(*
SPDX-FileCopyrightText: © 2026 Oleksandr Tiutyk <trofimich@gmail.com>
SPDX-License-Identifier: MIT
License: https://opensource.org/license/mit
*)

(*!
<summary>Loads file contents through cyclic task execution.</summary>
<description>
The native FB_FileLoad opens the file in binary mode, reads the requested byte count and closes it. Its
documented path support is the addressed target's local filesystem, not a network-share path. Use one owner
task. Configure FilePath, AmsNetId, TargetBuffer, TargetBufferSize and Timeout before Start and keep them
unchanged until STOPPED. The caller supplies live writable memory of at least TargetBufferSize bytes and
retains it through stopping after failure or cancellation. Do not access that memory concurrently with the
operation. Missing path, null buffer and zero size are rejected during execution; capacity and pointer
lifetime cannot be verified by this wrapper. Native errors use Task failure handling. Continue Execute until
STOPPED. Cancellation drains pending work without restoring buffer contents. WORK_DONE means the native
request completed without an error; this wrapper does not compare the returned byte count with file size or
promise a complete snapshot of a concurrently modified file. LoadedBytesCount exposes the result only after
STOPPED and WORK_DONE. Reset preserves configuration.
</description>
*)

{attribute 'no_explicit_call' := 'do not call this function block directly'}
FUNCTION_BLOCK LoadFile EXTENDS TOF_Tasks.Task IMPLEMENTS IFileSystemTask
VAR_STAT
	//! <summary>Static type metadata available before the base task initializes its default name.</summary>
	{attribute 'hide'}
	_ClassName : STRING := __POUNAME();
END_VAR
VAR
    _LoadFile : Tc2_System.FB_FileLoad; 
END_VAR

(*!
<summary>Selects the ADS target for the native filesystem operation.</summary>
<description>
Configure before Start and keep unchanged until STOPPED; the setter stores configuration without submitting
I/O.
</description>
*)
{attribute 'monitoring' := 'call'}
PROPERTY AmsNetId : Tc2_System.T_AmsNetID
GET
AmsNetId := _LoadFile.sNetId;
END_GET
SET
_LoadFile.sNetId := AmsNetId;
END_SET
END_PROPERTY

(*!
<summary>Provides the concrete type name used in diagnostics.</summary>
<description>
Returns borrowed read-only metadata; keep the instance alive and do not modify the referenced string.
Initialized static storage is ready during base Task.FB_init; this getter has no side effects or exceptions.
</description>
*)
{attribute 'monitoring' := 'call'}
PROPERTY ClassName : REFERENCE TO STRING
GET
ClassName REF= _ClassName;
END_GET
END_PROPERTY

(*!
<summary>Provides the configured path for the file operation.</summary>
<description>
The setter copies text without performing I/O. Configure before Start and keep unchanged until STOPPED; Reset
preserves it. The native service determines whether the path is usable.
</description>
*)
{attribute 'monitoring' := 'call'}
PROPERTY FilePath : Tc2_System.T_MaxString
GET
FilePath := _LoadFile.sPathName;
END_GET
SET
_LoadFile.sPathName := FilePath;
END_SET
END_PROPERTY

(*!
<summary>Reports the byte count from a successfully completed load.</summary>
<description>
Returns the native result only while State.Stopped and FinalStopReason.WorkDone are both TRUE. In every other
state, including READY, RUNNING, failure and cancellation, returns the initial value of the property type.
This default is not a success indicator; inspect the task state and final reason. Zero outside successful
completion does not mean the target buffer was unchanged. The getter does not modify native outputs or
buffers. Copy a successful result before Reset or reuse.
</description>
*)
{attribute 'monitoring' := 'call'}
PROPERTY LoadedBytesCount : UDINT
GET
IF NOT State.Stopped OR_ELSE NOT FinalStopReason.WorkDone THEN
	RETURN;
END_IF

LoadedBytesCount := _LoadFile.cbRead;
END_GET
END_PROPERTY

(*!
<summary>Provides the library namespace used in diagnostics.</summary>
<description>Returns borrowed read-only namespace storage; do not modify the referenced string.</description>
*)
{attribute 'monitoring' := 'call'}
PROPERTY NamespaceName : REFERENCE TO STRING
GET
NamespaceName REF= CurrentNamespace.Name;
END_GET
END_PROPERTY

(*!
<summary>Resets the native request edge after the task has stopped.</summary>
<description>
Preserves configured inputs and does not undo completed filesystem effects. Pending I/O must finish during
stopping before this hook runs.
</description>
*)
METHOD PROTECTED OnReset
_LoadFile(bExecute := FALSE);
END_METHOD

(*!
<summary>Submits and advances a native file load into caller-owned memory.</summary>
<description>
Validates required configuration before submitting the request. Native errors raise an exception for the base
Task failure/stopping path without dynamic string-builder allocations. Normal completion reports DONE only
after the native block is no longer busy. No rollback is performed.
</description>
<param name="processingState">BUSY while pending; DONE after native completion without an error.</param>
<param name="stopReasonMessage">Not changed here; failures are passed through exceptions.</param>
*)
METHOD PROTECTED OnRunning
VAR_OUTPUT
	processingState : TOF_Tasks.TASK_PROCESSING_STATE;
END_VAR
VAR_IN_OUT
	stopReasonMessage : TOF_Core.ERROR_MESSAGE;
END_VAR
VAR
	formattedExceptionMessage : TOF_Core.ERROR_MESSAGE;
END_VAR
IF NOT _LoadFile.bExecute THEN 
	IF TOF_Core.Strings.IsNullOrWhiteSpace(stringToCheck := _LoadFile.sPathName) THEN
		TOF_Core.Exceptions.ThrowDataMemberNotSpecified(
			sourceNamespaceName := NamespaceName,
			sourceClassName := ClassName,
			sourcePOUName := __POUNAME(),
			sourcePosition := __POSITION(),
			dataMemberName := 'FilePath'
		);		
	END_IF

	IF _LoadFile.pReadBuff = 0 THEN
		TOF_Core.Exceptions.ThrowDataMemberNotSpecified(
			sourceNamespaceName := NamespaceName,
			sourceClassName := ClassName,
			sourcePOUName := __POUNAME(),
			sourcePosition := __POSITION(),
			dataMemberName := 'TargetBuffer'
		);		
	END_IF

	IF _LoadFile.cbReadLen = 0 THEN
		TOF_Core.Exceptions.ThrowDataMemberNotSpecified(
			sourceNamespaceName := NamespaceName,
			sourceClassName := ClassName,
			sourcePOUName := __POUNAME(),
			sourcePosition := __POSITION(),
			dataMemberName := 'TargetBufferSize'
		);		
	END_IF
END_IF

_LoadFile(bExecute := TRUE);

IF _LoadFile.bError THEN
	TOF_Core.WideStrings.Append255(
		formattedExceptionMessage,
		"An error occurred while loading the file '",
		TO_WSTRING(_LoadFile.sPathName),
		"'");

	FileSystemExceptions.ThrowFileSystem(
		sourceNamespaceName := NamespaceName,
		sourceClassName := ClassName,
		sourcePOUName := __POUNAME(),
		sourcePosition := __POSITION(),
		message := formattedExceptionMessage,
		errorCode := _LoadFile.nErrId
	);
END_IF

IF NOT _LoadFile.bBusy THEN
	processingState := TOF_Tasks.TASK_PROCESSING_STATE.DONE;
END_IF
END_METHOD

(*!
<summary>Waits for an already submitted operation before task termination.</summary>
<description>
Runs for every stop reason. Advances the pending FB with bExecute=FALSE without issuing another request.
Completion does not roll back side effects. Keep configuration and borrowed buffers valid until STOPPED.
</description>
<param name="readyToRelease">TRUE when the underlying FB is no longer busy.</param>
*)
METHOD PROTECTED OnStopping
VAR_OUTPUT
	readyToRelease : BOOL;
END_VAR
IF _LoadFile.bBusy THEN
	_LoadFile(bExecute := FALSE);
END_IF

readyToRelease := NOT _LoadFile.bBusy;
END_METHOD

(*!
<summary>Reports the size of this concrete instance in bytes.</summary>
*)
{attribute 'monitoring' := 'call'}
PROPERTY SelfSize : ULINT
GET
SelfSize := XSIZEOF(THIS^);
END_GET
END_PROPERTY

(*!
<summary>Specifies the caller-owned writable buffer for loading file bytes.</summary>
<description>
Provide at least TargetBufferSize bytes and retain the buffer until STOPPED, including after cancellation or
failure. Null is rejected during execution. The wrapper cannot validate actual capacity or lifetime. Do not
access the buffer concurrently. Failure does not restore previous contents.
</description>
*)
{attribute 'monitoring' := 'call'}
PROPERTY TargetBuffer : POINTER TO BYTE
GET
TargetBuffer := _LoadFile.pReadBuff;
END_GET
SET
_LoadFile.pReadBuff := TargetBuffer;
END_SET
END_PROPERTY

(*!
<summary>Specifies the positive number of bytes requested from the file.</summary>
<description>
Passed to native cbReadLen. Must not exceed the caller-owned TargetBuffer capacity. Zero is rejected during
execution and identifies TargetBufferSize in the failure diagnostic. Keep this value unchanged from Start
through STOPPED. LoadedBytesCount reports the actual count only after successful completion; this setting does not assert that the entire file fits in the buffer.
</description>
*)
{attribute 'monitoring' := 'call'}
PROPERTY TargetBufferSize : UDINT
GET
TargetBufferSize := _LoadFile.cbReadLen;
END_GET
SET
_LoadFile.cbReadLen := TargetBufferSize;
END_SET
END_PROPERTY

(*!
<summary>Configures the timeout passed to native operation requests.</summary>
<description>
Set before Start and keep unchanged until STOPPED. Reset preserves this value. It is not an overall task
deadline or a guarantee of resource release after a timeout.
</description>
*)
{attribute 'monitoring' := 'call'}
PROPERTY Timeout : TIME
GET
Timeout := _LoadFile.tTimeout;
END_GET
SET
_LoadFile.tTimeout := Timeout;
END_SET
END_PROPERTY

END_FUNCTION_BLOCK

(* stored: Version 1.1.0.1
   POU LoadFile: Id {f209aa42-7adf-492c-aad8-55961c90382f}, SpecialFunc None
   Folder Inputs: Id {18728b97-c728-45b7-bb38-dbaf4d4aab74}
   Folder Members to override: Id {6ce189b7-b717-41ff-9d6c-3f28fa29db0f}
   Folder Outputs: Id {b1a24ae9-9d25-4f51-a8dd-c308ec8de3dd}
   Property AmsNetId: Id {af068792-c8f4-4f1a-a44a-adda9d288f6d}
   Get Get: Id {868a196a-7436-448f-9a7e-6fd1d69498cf}
   Set Set: Id {d19a998d-9017-4398-9524-9da7a5394778}
   Property ClassName: Id {96970123-0d8d-47e6-83f1-a38f9bb70154}
   Get Get: Id {c4ee9f16-700c-4449-bcc0-45c65b7ac32a}
   Property FilePath: Id {df0a29d4-2663-49ed-9a38-1172e5e4cc52}
   Get Get: Id {1fad573b-82ff-449a-86bd-730b2a3e7f22}
   Set Set: Id {d5449e43-882b-4573-8365-1f36f6161f08}
   Property LoadedBytesCount: Id {54d91487-d011-40f7-9d29-569f0b2da1c8}
   Get Get: Id {f1c7a567-7f12-4f86-9023-1a9d28698d04}
   Property NamespaceName: Id {a88dba22-63c9-49ea-8020-f00da78e287e}
   Get Get: Id {3f934858-f9ad-49d7-b681-cddd5e0528f3}
   Method OnReset: Id {5681e281-0f75-465c-88ec-d9a447202e30}
   Method OnRunning: Id {03e4a860-0585-482d-b55c-424c8666832b}
   Method OnStopping: Id {6a92da47-266c-4f5c-89b8-935661f5c451}
   Property SelfSize: Id {a442a130-81b3-4e43-b979-44693957f557}
   Get Get: Id {bdc789ba-8674-416a-98ce-60346ba17014}
   Property TargetBuffer: Id {9dd63f9e-2d64-461f-a3f5-07ac6784c88a}
   Get Get: Id {2a072640-ef4c-41ce-8e43-473c69610ee4}
   Set Set: Id {9a9aecdb-7c7d-488c-a57d-91bd8e872383}
   Property TargetBufferSize: Id {c19ac729-8465-479e-a11f-bb4a5d725ea5}
   Get Get: Id {a1b09fc4-82e3-4916-a73f-f250bd341d13}
   Set Set: Id {bb7c677e-68c6-4d91-bcd8-d7df9490f3d3}
   Property Timeout: Id {2e18453b-9571-436c-b47d-3e985ed694df}
   Get Get: Id {efd36739-8d02-40db-be47-4114d401c9d1}
   Set Set: Id {a7b1d0e6-8ec9-4ee8-95b8-368aea4595b6} *)
